# EPICS autosave request: ADAndorIstar/andorIstarApp/Db/andorIstar_settings.req
$(P)$(R)AndorCooler
$(P)$(R)Temperature
$(P)$(R)TriggerMode
$(P)$(R)ImageMode
$(P)$(R)AndorReadMode
$(P)$(R)AndorGateMode
$(P)$(R)AcquireTime
$(P)$(R)AndorDDGGateWidth
$(P)$(R)AndorDDGGateDelay
$(P)$(R)AndorDDGIOC
$(P)$(R)AndorMCPGain
$(P)$(R)AndorPreAmpGain
$(P)$(R)AndorADCSpeed
$(P)$(R)FitsHeaderFileName
$(P)$(R)DataType
$(P)$(R)ArrayCallbacks
$(P)$(R)PALFilePath
